// Mitsubishi GX Works2 project: test   PLC: FX3U/FX3UC

// task Task_01 (event TRUE, interval 0, priority 31): POU_01

PROGRAM POU_01
VAR
  map : ARRAY [0..24] OF INT;
  ii : INT;
  isum_Q : INT;
  isum_A : INT;
  rand_seed : INT;
  R_TRIG_start : R_TRIG;
  wstep : INT;
  TON_timer : TON;
  TON_start : TON;
  TON_end : TON;
  TON_reset : TON;
END_VAR
(*
M0~M24 按鈕
D0~D24 數字顯示 (含背光)

M90 開始按鈕
D90 計時器
D91 關卡數
D92 狀態顯示 (wstep)
D93 目標關卡
D94 顯示快慢
D95 猜測快慢
D96 輸贏
D97 按鈕燈號
*)

R_TRIG_start(_CLK := M90); (*開始按鈕上緣*)
D8000 := 1000; (*看門狗設定為 1 秒*)
D92 := wstep; (*將wstep搬至 D92*)

(*開機*)
IF M8002 THEN
	D93 := 5;
	D94 := 3;
	D95 := 3;
	D85 := 3;
	wstep := 0;
END_IF;
(*重置*)
TON_reset(IN := M90, PT := T#1s);
IF TON_reset.Q THEN
	wstep := 0;
END_IF;

CASE wstep OF
	0: (*初始狀態*)
	D97 := 0;
	
	(*亂數種子*)
	rand_seed := rand_seed + 1;
	IF rand_seed > 30000 THEN
		rand_seed := 0;
	END_IF;
	
	(*復歸*)
	ZRST(TRUE, D0, D24);
	ZRST(TRUE, D90, D91);
	
	(*當按下開始按鈕*)
	IF R_TRIG_start.Q AND (D93 <> 0) THEN
		D90 := 30;
		wstep := 20;
	END_IF;
	
	20: (*遊戲開始*)
	(*倒數 3秒 開始*)
	TON_start(IN := NOT TON_start.Q, PT := T#0.1s);
	IF TON_start.Q THEN
		D90 := D90 - 1;
	END_IF;
	
	(*倒數結束*)
	IF D90 = 0 THEN
		D90 := 20; 
		isum_Q := 0; (*第一關*)
		map := rand(rand_seed); (*產數亂數*)
		wstep := 21;
	END_IF;	
	
	21: (*顯示數字*)
	D91 := isum_Q + 1; (*顯示關卡*)
	FOR ii := 0 TO isum_Q BY 1 DO
		map[ii] := map[ii] MOD 25;	(*限制亂數範圍*)
		
		(*數字*)
		Z1 := map[ii];
		D0Z1 := ii + 2;
	END_FOR;
	
	(*倒數計時*)
	TON_timer(IN := NOT TON_timer.Q, PT := T#0.1s);
	IF TON_timer .Q THEN
		D90 := D90 - 1;
	END_IF;	
	(*倒數結束*)
	IF D90 <= 0 THEN
		
		(*清數字顯示*)
		FOR ii := 0 TO 24 BY 1 DO
			Z2 := ii;
			IF D0Z2 <> 0 THEN
				D0Z2 := 1;
			END_IF;
		END_FOR;
		D90 := (15 + ((isum_Q/D95) * 10)); (*設定猜測計時*)
		isum_A := 1;
		wstep := 22;
	END_IF;		
	
	22:
	(*猜測按鈕*)
	FOR ii := 0 TO 24 BY 1 DO
		Z3 := ii;			
		
		(*遊玩按鈕*)
		IF M0Z3 AND (D0Z3 = 1) THEN (*按下按鈕 且 有背光*)
			IF map[isum_A - 1] =  ii THEN (*按下正確的按鈕順序*)
				isum_A := isum_A + 1;
				D0Z3 := 0;
			ELSE
				wstep := 30;
			END_IF; 
		END_IF;
		
		(*當全部猜完*)
		IF isum_A = isum_Q + 2 THEN
			isum_Q := isum_Q + 1;
			D90 := 15 + ((isum_Q / D94) * 10); (*重新設定顯示時間*)

			(*產生亂數*)
			rand_seed := map[24] + map[23];
			IF rand_seed > 30000 THEN
				rand_seed := 0;
			END_IF;
			map := rand(rand_seed);

			(*贏的條件*)
			IF isum_Q >= D93 THEN
				wstep := 40;
			ELSE
				wstep := 21;
			END_IF;
		END_IF;
	END_FOR;
	
	(*倒數計時*)
	TON_timer(IN := NOT TON_timer.Q, PT := T#0.1s);
	IF TON_timer .Q THEN
		D90 := D90 - 1;
	END_IF;	
	(*倒數結束*)
	IF D90 <= 0 THEN
		wstep := 30;
	END_IF;	
	
	30:
	(*計時3秒*)
	TON_end(IN := NOT TON_end.Q, PT := T#3s);
	IF TON_end.Q THEN
		wstep := 31;
	END_IF;	
	
	(*顯示未按的按鈕*)	
	FOR ii := 0 TO 24 BY 1 DO
		Z4 := map[ii];
		IF D0Z4 = 1 THEN
			D0Z4 := isum_A;
			isum_A := isum_A + 1;
		END_IF;  
	END_FOR;
	
	31:
	D96 := 1;
	(*計時3秒*)
	TON_end(IN := NOT TON_end.Q, PT := T#3s);
	IF TON_end.Q THEN
		wstep := 0;
	END_IF;		
	
	40:
	D96 := 2;
	(*計時3秒*)
	TON_end(IN := NOT TON_end.Q, PT := T#3s);
	IF TON_end.Q THEN
		wstep := 0;
	END_IF;		
	
END_CASE;
END_PROGRAM

FUNCTION rand
VAR_INPUT
  seed : INT;
END_VAR
VAR
  result : ARRAY [0..24] OF INT;
  ii : INT;
  ij : INT;
END_VAR
result[0] :=  ABS( (D8013 + D8014 + D8015)  * D8016 + seed + D8010) MOD 20021; (*第一亂數*)

FOR ii := 0 TO 24 BY 1 DO
	RCL(TRUE, 37, result[ii]);
	result[ii + 1] := ABS( (result[ii] + 1853) ) MOD 15061; (*線性同餘法*)
END_FOR;
rand := result;
END_FUNCTION
